Xinje XDPPro project, PLC1: RC2V6 (software 3.3 2016-03-11)

PROGRAM Ladder

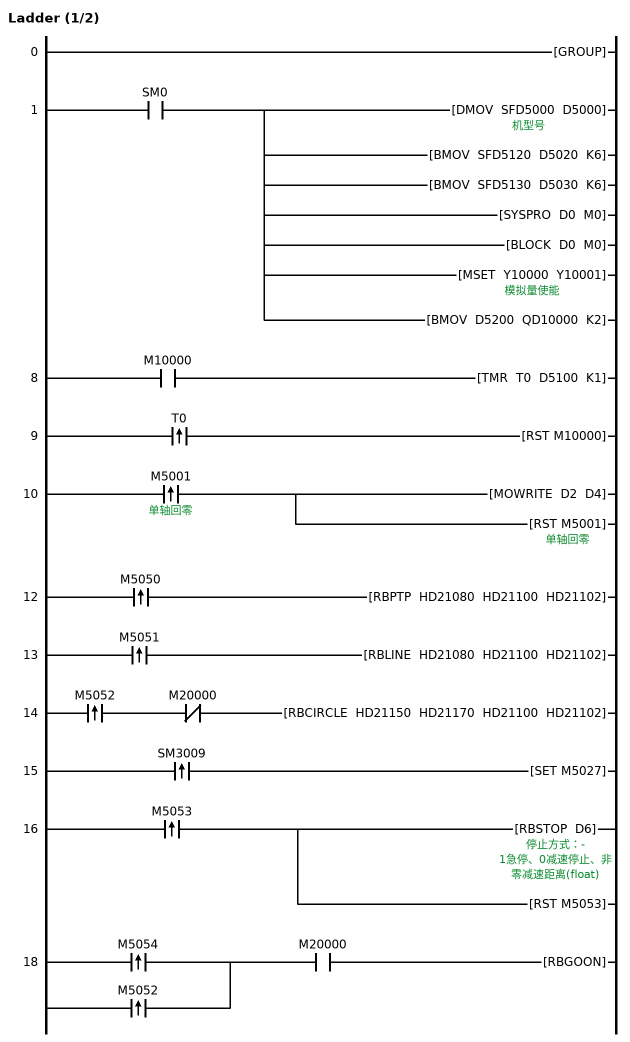
GROUP
LD     SM0
DMOV   SFD5000 D5000	; 机型号
BMOV   SFD5120 D5020 K6
BMOV   SFD5130 D5030 K6
SYSPRO D0 M0
BLOCK  D0 M0
MSET   Y10000 Y10001	; 模拟量使能
BMOV   D5200 QD10000 K2
LD     M10000
TMR    T0 D5100 K1
LDP    T0
RST    M10000
LDP    M5001	; 单轴回零
MOWRITE D2 D4
RST    M5001	; 单轴回零
LDP    M5050
RBPTP  HD21080 HD21100 HD21102
LDP    M5051
RBLINE HD21080 HD21100 HD21102
LDP    M5052
ANI    M20000
RBCIRCLE HD21150 HD21170 HD21100 HD21102
LDP    SM3009
SET    M5027
LDP    M5053
RBSTOP D6	; 停止方式：-1急停、0减速停止、非零减速距离(float)
RST    M5053
LDP    M5054
ORP    M5052
AND    M20000
RBGOON

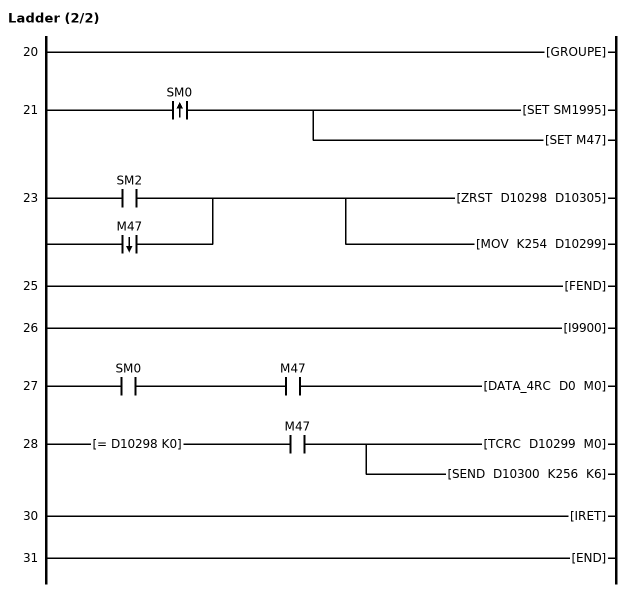
GROUPE
LDP    SM0
SET    SM1995
SET    M47
LD     SM2
ORF    M47
ZRST   D10298 D10305
MOV    K254 D10299
FEND
I9900
LD     SM0
AND    M47
DATA_4RC D0 M0
LD=    D10298 K0
AND    M47
TCRC   D10299 M0
SEND   D10300 K256 K6
IRET
END

COMMENTS (devices not used above)
M5040	PTP运动标志
HD0	shang
HD20	xia
HD40	chang
HD60	zhong
HD110	.

C FUNCTION BLOCK block.fcb
/*************************************************************************
   FunctionBlockName:  BLOCK
   Version:            1.0.0
   Author:             
   UpdateTime:         2016/6/1 9:27:03
   Comment:            
			20161123：RBON
**************************************************************************/
#define SysRegAddr_HD_SD_FD_SM_HSD_Y_X_D
#define PT_SIZE_WD          20
#define INT_BEGADDR_HD(i)   (10+i*2)       //200个int变量(10~309)
#define FLOAT_BEGADDR_HD(i) (410+i*2)      //200个float变量(410~809) 
#define POINT_BEGADDR_HD(i) (1000+i*PT_SIZE_WD)
#define Decimal_HEX(i)      (i-i/10*2)
#define SysModelType    X[26]          //0手动、1自动

//FUNC CODE
#define IF_BIT    1004
#define END_IF    1005
#define WAIT      1006
#define SET       1007
#define RESET     1008
#define IF_VALUE  1044
#define DELAY_MM  1003
#define LOOP      1009
#define END_LOOP  1010
#define WHILE     1011
#define END_WHILE 1012
#define LABLE     1013
#define GOTO      1014
#define ASSIGN    1020
#define PTASSIGN  1021
#define OFST      1022
#define SETACC    1023
#define CALL      1050
#define PTP       1030
#define MOVL      1031
#define MOVC      1032
#define WELD      1040
#define END_WELD  1041

#define MAINPRO_SIZE HD[3000]
#define SUBPRO1_SIZE HD[3001]
#define SUBPRO2_SIZE HD[3002]
#define SUBPRO3_SIZE HD[3003]
#define SUBPRO4_SIZE HD[3004]
#define TASK1_SIZE  HD[3005]
#define TASK2_SIZE  HD[3006]
#define proBlockSize(i) HD[3000+i]
#define SUBPRO_TOTAL_SIZE_WD 2000
#define FUNCCODE_SIZE_WD    20
#define MAINPRO_BEGADDR_HD  3020
#define SUBPRO_BEGADDR_HD   9020
#define curRunProIndex     HD[21040]
#define runRow_CurIndex(i) HD[21050+i]
#define runRow_UpIndex(i)  HD[21060+i]

#define X_BASE_BEGADDR  2140000000
#define Y_BASE_BEGADDR  2141000000
#define M_BASE_BEGADDR  2142000000
#define CHECK_X(index)  (index>=X_BASE_BEGADDR && index<=2140000099)
#define CHECK_Y(index)  (index>=Y_BASE_BEGADDR && index<=2141000199)
#define CHECK_M(index)  (index>=M_BASE_BEGADDR && index<=2142002999)

#define PRO_SINGLE_STEP_M 5025
#define PRO_RUN_M         5026
#define MOVE_END_FLAG     5027

#define PTP_TRIG_SINGAL_M    5050
#define MOVL_TRIG_SINGAL_M   5051
#define MOVC_TRIG_SINGAL_M   5052
#define ROBOT_RUNSTOP_M      5024

#define PT_BEGADDR_HD        21080
#define MOVSPEED_BEGADDR_HD  21100
#define MOVC_PT_BEGADDR_HD   21150
#define MOVC_PT_ENDADDR_HD   21170

#define ROBOT_ON   SM[3000]
#define RBRUN_ON   SM[3001]
#define ALARM_FLAG SM[3004]
#define WARN_FLAG  SM[3005]

#define ACCDEF_VALUE 70
#define SETACC_VALUE *(float*)&HD[21102]

float userSetAcc = 0;
int tmrVal=0;
int funcBegAddr_HD = 0;
int flag = 0,flag1=0;
extern int funcCodeRunFlag;
void funcExplanPro(BIT B,WORD W,int proIndex,int funcBegAddr_HD);
void IF_BIT_Pro(WORD W,BIT B,int pIndex);
void END_IF_Pro(int pIndex);
void DELAY_Pro(BIT B,WORD W,int proIndex);
void WAIT_Pro(BIT B,WORD W,int proIndex);
void SET_Pro(BIT B,int pIndex);
void RESET_Pro(BIT B,int pIndex);
void LOOP_Pro(int pIndex);
void END_LOOP_Pro(int pIndex);
void WHILE_Pro(WORD W,BIT B,int pIndex);
void END_WHILE_Pro(int pIndex);
void ASSIGN_Pro(WORD W,int pIndex);
void PTASSIGN_Pro(WORD W,int pIndex);
void OFST_Pro(WORD W,int pIndex);
void SETACC_Pro(WORD W,BIT B,int proIndex);
void GOTO_Pro(int pIndex);
void CALL_Pro();
void PTP_MOVL_Pro(BIT B,int proIndex);
void MOVC_Pro(BIT B,int proIndex);
void WELD_Pro(WORD W,BIT B,int proIndex);
void END_WELD_Pro(WORD W,BIT B,int proIndex);

#define RUNINDEX_PRO(proIndex){runRow_UpIndex(proIndex) = runRow_CurIndex(proIndex);\
					 runRow_CurIndex(proIndex)++;\
					 funcCodeRunFlag = 0;}

void BLOCK( WORD W , BIT B )
{
#define SysRegAddr_HD_SD_FD_SM_HSD_Y_X
#define DHD *(int*)&HD
#define FHD *(float*)&HD

	int i;
//B[10]=funcCodeRunFlag;
//B[11]=flag;
//B[12]=flag1;
	B[5056]=funcCodeRunFlag;
	if(userSetAcc==0)
		userSetAcc = ACCDEF_VALUE;	
	for(i=0; i<7; i++)
	{
		if(runRow_CurIndex(i)==0)
		{
			runRow_CurIndex(i)=1;
			flag = 0,flag1=0,funcCodeRunFlag = 0;
		}
	}
	if(ROBOT_ON==0||ALARM_FLAG==1||WARN_FLAG==1)
	{
		B[PTP_TRIG_SINGAL_M]=0;
		B[MOVL_TRIG_SINGAL_M]=0;
		B[MOVC_TRIG_SINGAL_M]=0;
		B[PRO_RUN_M]=0;
		flag = 0,flag1=0,funcCodeRunFlag = 0;
		B[MOVE_END_FLAG]=SM[3009];
		B[10000]=0;
		B[20000]=0;
		B[20001]=0;
		return;
	}
	if((B[PRO_SINGLE_STEP_M]==1||B[PRO_RUN_M]==1)&&B[20001]==1)
    	B[20001]=0;//清除圆弧未完成停止辅助信号
	if(runRow_CurIndex(curRunProIndex)<=proBlockSize(curRunProIndex)&&ALARM_FLAG==0)
	{
		if((B[PRO_SINGLE_STEP_M]==1||B[PRO_RUN_M]==1)&&funcCodeRunFlag==0)//下一步
		{
			funcCodeRunFlag=1;
			B[PRO_SINGLE_STEP_M]=0;
		}
	}
	if(funcCodeRunFlag==1)
	{
		funcBegAddr_HD = MAINPRO_BEGADDR_HD+(runRow_CurIndex(0)-1)*FUNCCODE_SIZE_WD;
		funcExplanPro(B,W,0,funcBegAddr_HD);
	}
}

void funcExplanPro(BIT B,WORD W,int proIndex,int funcBegAddr_HD)
{
	switch(HD[funcBegAddr_HD])
	{
	case IF_BIT:
		IF_BIT_Pro(W,B,proIndex);
		break;
	case END_IF:
		END_IF_Pro(proIndex);
		break;
	case DELAY_MM:
		DELAY_Pro(B,W,proIndex);
		break;
	case WAIT:
		WAIT_Pro(B,W,proIndex);
		break;
	case SET:
		SET_Pro(B,proIndex);
		break;
	case RESET:
		RESET_Pro(B,proIndex);
		break;
	case LOOP:
		LOOP_Pro(proIndex);
		break;
	case END_LOOP:
		END_LOOP_Pro(proIndex);
		break;
	case WHILE:
		WHILE_Pro(W,B,proIndex);
		break;
	case END_WHILE:
		END_WHILE_Pro(proIndex);
		break;
	case ASSIGN:
		ASSIGN_Pro(W,proIndex);
		break;
	case PTASSIGN:
		PTASSIGN_Pro(W,proIndex);
		break;
	case OFST:
		OFST_Pro(W,proIndex);
		break;
	case SETACC:
		SETACC_Pro(W,B,proIndex);
		break;	
	case LABLE:
		funcCodeRunFlag=0;
		runRow_UpIndex(proIndex) = runRow_CurIndex(proIndex);
		runRow_CurIndex(proIndex)++;
		break;
	case GOTO:
		GOTO_Pro(proIndex);
		break;
	case CALL:
		curRunProIndex = HD[funcBegAddr_HD+1];		
		CALL_Pro(B,W);
		break;
	case PTP:
		PTP_MOVL_Pro(B,proIndex);
		break;
	case MOVL:
		PTP_MOVL_Pro(B,proIndex);
		break;
	case MOVC:
		MOVC_Pro(B,proIndex);
		break;
	case WELD:
		WELD_Pro(W,B,proIndex);
		break;	
	case END_WELD:
		END_WELD_Pro(W,B,proIndex);
		break;	
	default:
		break;
	}
}

BOOL GetBitStatu(int bitAddr,BIT B)
{
	BOOL rlt=0;
	if(CHECK_X(bitAddr))
	{
		rlt = X[Decimal_HEX((bitAddr-X_BASE_BEGADDR))];
	}
	else if(CHECK_Y(bitAddr))
	{
		rlt = Y[Decimal_HEX((bitAddr-Y_BASE_BEGADDR))];
	}
	else if(CHECK_M(bitAddr))
	{
		rlt = B[bitAddr-M_BASE_BEGADDR];
	}
	return rlt;
}

BOOL GetBitCaseValue(BIT B,int begAddr)
{
	char cmpVal = 0;
	int para1 = DHD[begAddr+2],para2 = DHD[begAddr+4];
	int para3 = DHD[begAddr+6],para4 = DHD[begAddr+8];
	int para5 = DHD[begAddr+10],para6 = DHD[begAddr+12];
	int para7 = DHD[begAddr+14];
	
	cmpVal = GetBitStatu(para1,B);
	if(para2!=0)
	{
		if(para2==1)
			cmpVal = cmpVal|GetBitStatu(para3,B);
		else
			cmpVal = cmpVal&GetBitStatu(para3,B);
		if(para4!=0)
		{
			if(para4==1)
				cmpVal = cmpVal|GetBitStatu(para5,B);
			else
				cmpVal = cmpVal&GetBitStatu(para5,B);
			if(para6!=0)
			{
				if(para6==1)
					cmpVal = cmpVal|GetBitStatu(para7,B);
				else
					cmpVal = cmpVal&GetBitStatu(para7,B);
			}
		}
	}
	return cmpVal;
}

BOOL GetWordCompareResult(WORD W,int begAddr)
{
	char i,cmpVal = 0;
	float cmp[2]= {0};

	for(i=0; i<2; i++)
	{
		if(DHD[begAddr+4+i*6]==1)      //W
			cmp[i] = DHD[INT_BEGADDR_HD(DHD[begAddr+6+i*6])];
		else if(DHD[begAddr+4+i*6]==2) //F
			cmp[i] = FHD[FLOAT_BEGADDR_HD(DHD[begAddr+6+i*6])];
		else
			cmp[i] = FHD[begAddr+6+i*6];
	}
	if(DHD[begAddr+8]==1)
		cmpVal = (cmp[0]>cmp[1]);
	else if(DHD[begAddr+8]==2)
		cmpVal = (cmp[0]>=cmp[1]);
	else if(DHD[begAddr+8]==3)
		cmpVal = (cmp[0]<cmp[1]);
	else if(DHD[begAddr+8]==4)
		cmpVal = (cmp[0]<=cmp[1]);
	else if(DHD[begAddr+8]==5)
		cmpVal = (cmp[0]==cmp[1]);
	else if(DHD[begAddr+8]==6)
		cmpVal = (cmp[0]!=cmp[1]);
	return cmpVal;
}

void Set_Reset_Bit(BIT B,int addr,int value)
{
	int para1 = DHD[addr+2],para2 = DHD[addr+4];
	int i,index1,index2;
	if(CHECK_Y(para1))
	{
		index1 = para1-Y_BASE_BEGADDR;
		Y[Decimal_HEX(index1)]=value;
	}
	else if(CHECK_M(para1))
	{
		index1 = para1-M_BASE_BEGADDR;
		B[index1]=value;
	}
	if(para2!=0)
	{
		if(CHECK_Y(para2))
		{
			index2 = para2-Y_BASE_BEGADDR;
			for(i=0; i<(index2-index1+1); i++)
				Y[Decimal_HEX((index1+i))]=value;
		}
		else if(CHECK_M(para2))
		{
			index2=para2-M_BASE_BEGADDR;
			for(i=0; i<(index2-index1+1); i++)
				B[index1+i]=value;
		}
	}
}
float GetAssignPara(int type,int index,int addr)
{
	float val = 0;
	if(type==1)     //W
		val=DHD[INT_BEGADDR_HD(index)];
	else if(type==2)//F
		val=FHD[FLOAT_BEGADDR_HD(index)];
	else              //K
		val=FHD[funcBegAddr_HD+addr];
	return val;
}
float CalcAssignResult(int operateType,float para1,float para2)
{
	float val=0;
	if(operateType==1)
		val=para1+para2;
	else if(operateType==2)
		val=para1-para2;
	else if(operateType==3)
		val=para1*para2;
	else if(operateType==4)
		val=para1/para2;
	else
		val = para1;
	return val;
}

void DELAY_Pro(BIT B,WORD W,int proIndex)
{
	int type = HD[funcBegAddr_HD+1];
	if(flag==0)
	{
		if(type==0)
			DW[5100]=DHD[funcBegAddr_HD+2];
		else
			DW[5100]=DHD[INT_BEGADDR_HD(HD[funcBegAddr_HD+2])];
		if(DW[5100]!=0)
		{
			flag = 1;
			B[10000]=1;
		}
		else
		{
			flag = 0;
			funcCodeRunFlag=0;
			B[10000]=0;
		}
	}
	else if(flag==1&&B[10000]==0)
	{
		flag = 0;
		RUNINDEX_PRO(proIndex)
	}
}

void IF_BIT_Pro(WORD W,BIT B,int proIndex)
{
	BOOL tmpBL = 0;
	if(DHD[funcBegAddr_HD+2]>=X_BASE_BEGADDR)
		tmpBL = GetBitCaseValue(B,funcBegAddr_HD);
	else
		tmpBL=GetWordCompareResult(W,funcBegAddr_HD);

	if(tmpBL==1)
	{
		RUNINDEX_PRO(proIndex)
	}
	else
	{
		int j,cycNum = proBlockSize(proIndex)-runRow_CurIndex(proIndex);
		for(j=0; j<cycNum; j++)
		{
			int tmpFuncCode = HD[funcBegAddr_HD+(j+1)*FUNCCODE_SIZE_WD];
			int endFlag = HD[funcBegAddr_HD+(j+1)*FUNCCODE_SIZE_WD+1];
			if(tmpFuncCode==END_IF&&endFlag==runRow_CurIndex(proIndex))
			{
				runRow_CurIndex(proIndex) = runRow_CurIndex(proIndex)+j+1;
				funcCodeRunFlag = 0;
				break;
			}
		}
	}
}
void END_IF_Pro(int proIndex)
{
	RUNINDEX_PRO(proIndex)
}

void WAIT_Pro(BIT B,WORD W,int proIndex)
{
	int timeType = DHD[funcBegAddr_HD+15],timeVal = DHD[funcBegAddr_HD+17];
	int fltTime = HD[funcBegAddr_HD+19],blTmp=0;
	int blrslt=0;
	int siglRslt = GetBitCaseValue(B,funcBegAddr_HD-1);
	
	if(timeType!=0)
		timeVal = DHD[INT_BEGADDR_HD(timeVal)];
	if(fltTime!=0&&siglRslt==1&&flag1==0)
	{		
		if(flag==1&&SM[11]==0)
			tmrVal++;
		flag = SM[11];
		if(tmrVal*5<fltTime)
			return;	
	}
	else
		flag1 = 1;
			
	if(timeVal!=0 && flag1==1 && flag==0)
	{
		DW[5100]=timeVal;
		B[10000]=1;	
		flag = 1;
	}
	if(timeVal!=0&&flag1==1&&B[10000]==0)
	{
		blTmp = 1;	
		flag = 0;
	}
	if(siglRslt==1 || blTmp==1)
	{
		RUNINDEX_PRO(proIndex)		
	}
	tmrVal = 0;
	flag1 = 0;
}
void SET_Pro(BIT B,int proIndex)
{
	Set_Reset_Bit(B,funcBegAddr_HD,1);
	RUNINDEX_PRO(proIndex)
}
void RESET_Pro(BIT B,int proIndex)
{
	Set_Reset_Bit(B,funcBegAddr_HD,0);
	RUNINDEX_PRO(proIndex)
}

void LOOP_Pro(int proIndex)
{
	int para1=DHD[funcBegAddr_HD+2],para2=DHD[funcBegAddr_HD+4];
	int loop_cycNum=0,begAddr=0;
	if(para1==0)
		loop_cycNum = para2;
	else
		loop_cycNum = DHD[INT_BEGADDR_HD(para2)];
	if(proIndex==0)
		begAddr=MAINPRO_BEGADDR_HD;
	else
		begAddr=SUBPRO_BEGADDR_HD;
	if(runRow_CurIndex(proIndex)>=runRow_UpIndex(proIndex))//||HD[begAddr+(runRow_UpIndex(proIndex)-1)*FUNCCODE_SIZE_WD]!=END_LOOP)
		DHD[funcBegAddr_HD+8]=0;

	if(loop_cycNum<=0)
	{
		int j,cycNum = proBlockSize(proIndex)-runRow_CurIndex(proIndex);
		for(j=0; j<cycNum; j++)
		{
			int tmpFuncCode = HD[funcBegAddr_HD+(j+1)*FUNCCODE_SIZE_WD];
			int endFlag = HD[funcBegAddr_HD+(j+1)*FUNCCODE_SIZE_WD+1];
			if(tmpFuncCode==END_LOOP&&endFlag==runRow_CurIndex(proIndex))
			{
				runRow_CurIndex(proIndex) = runRow_CurIndex(proIndex)+j+1;
				break;
			}
		}
	}
	else
	{
		DHD[funcBegAddr_HD+8]=DHD[funcBegAddr_HD+8]+1;
		RUNINDEX_PRO(proIndex)
	}
	funcCodeRunFlag = 0;
}
void END_LOOP_Pro(int proIndex)
{
	int para1=DHD[funcBegAddr_HD+1];
	int loop_BegAddr=0,loop_para1,loop_para2,curNum,loop_cycNum=0;
	if(proIndex==0)
		loop_BegAddr = MAINPRO_BEGADDR_HD+(para1-1)*FUNCCODE_SIZE_WD;
	else
		loop_BegAddr = SUBPRO_BEGADDR_HD+(proIndex-1)*SUBPRO_TOTAL_SIZE_WD+(para1-1)*FUNCCODE_SIZE_WD;

	loop_para1=DHD[loop_BegAddr+2];
	loop_para2=DHD[loop_BegAddr+4];
	curNum = DHD[loop_BegAddr+8];

	if(loop_para1==0)
		loop_cycNum = loop_para2;
	else
		loop_cycNum = DHD[INT_BEGADDR_HD(loop_para2)];

	runRow_UpIndex(proIndex) = runRow_CurIndex(proIndex);
	if(curNum==loop_cycNum)
	{
		DHD[loop_BegAddr+8]=0;
		runRow_CurIndex(proIndex)++;
	}
	else
		runRow_CurIndex(proIndex)=para1;
	funcCodeRunFlag = 0;
}
void WHILE_Pro(WORD W,BIT B,int proIndex)
{
	BOOL tmpBL = 0;
	if(DHD[funcBegAddr_HD+2]>=X_BASE_BEGADDR)
		tmpBL = GetBitCaseValue(B,funcBegAddr_HD);
	else
		tmpBL=GetWordCompareResult(W,funcBegAddr_HD);
	if(tmpBL==1)
	{
		RUNINDEX_PRO(proIndex)
	}
	else
	{
		int j,cycNum = proBlockSize(proIndex)-runRow_CurIndex(proIndex);
		for(j=0; j<cycNum; j++)
		{
			int tmpFuncCode = HD[funcBegAddr_HD+(j+1)*FUNCCODE_SIZE_WD];
			int endFlag = HD[funcBegAddr_HD+(j+1)*FUNCCODE_SIZE_WD+1];
			if(tmpFuncCode==END_WHILE&&endFlag==runRow_CurIndex(proIndex))
			{
				runRow_CurIndex(proIndex) = runRow_CurIndex(proIndex)+j+1+1;
				funcCodeRunFlag = 0;
				break;
			}
		}
	}
}
void END_WHILE_Pro(int proIndex)
{
	int para1=DHD[funcBegAddr_HD+1];

	runRow_UpIndex(proIndex) = runRow_CurIndex(proIndex);
	runRow_CurIndex(proIndex) = para1;
	funcCodeRunFlag = 0;
}

void ASSIGN_Pro(WORD W,int proIndex)
{
	int leftParaType = HD[funcBegAddr_HD+1],leftPara=HD[funcBegAddr_HD+2];

	int rightPara1Type = DHD[funcBegAddr_HD+4],rightPara1=DHD[funcBegAddr_HD+6];
	int operaFlag1 = DHD[funcBegAddr_HD+8];
	int rightPara2Type = DHD[funcBegAddr_HD+10],rightPara2=DHD[funcBegAddr_HD+12];
	int operaFlag2 = DHD[funcBegAddr_HD+14];
	int rightPara3Type = DHD[funcBegAddr_HD+16],rightPara3=DHD[funcBegAddr_HD+18];

	float result1,result;
	float para1=GetAssignPara(rightPara1Type,rightPara1,6);
	float para2=GetAssignPara(rightPara2Type,rightPara2,12);
	float para3=GetAssignPara(rightPara3Type,rightPara3,18);

	result1 = CalcAssignResult(operaFlag1,para1,para2);
	result = CalcAssignResult(operaFlag2,result1,para3);

	if(leftParaType==1)
		DHD[INT_BEGADDR_HD(leftPara)]=result;
	else if(leftParaType==2)
		FHD[FLOAT_BEGADDR_HD(leftPara)]=result;
	RUNINDEX_PRO(proIndex)
}

void PTASSIGN_Pro(WORD W,int proIndex)
{
	int targetPtType = HD[funcBegAddr_HD+1],targetPt=0;
	int basePtType =   HD[funcBegAddr_HD+3],basePt=0;
	int coordIndex =   HD[funcBegAddr_HD+5];
	int ofstValueType1 =HD[funcBegAddr_HD+7],ofstValue1=DHD[funcBegAddr_HD+8];
	int operaFlag1 = HD[funcBegAddr_HD+10];	
	int ofstValueType2 =HD[funcBegAddr_HD+11],ofstValue2=DHD[funcBegAddr_HD+12];
	float para1=0,para2=0,ofstValue=0;
	para1=GetAssignPara(ofstValueType1,ofstValue1,8);
	if(operaFlag1!=0)
		para2=GetAssignPara(ofstValueType2,ofstValue2,12);
	ofstValue = CalcAssignResult(operaFlag1,para1,para2);
	if(targetPtType==0)
		targetPt = HD[funcBegAddr_HD+2];
	else
		targetPt = DHD[INT_BEGADDR_HD(HD[funcBegAddr_HD+2])];
	if(basePtType==0)
		basePt = HD[funcBegAddr_HD+4];
	else
		basePt = DHD[INT_BEGADDR_HD(HD[funcBegAddr_HD+4])];			  		
	memcpy(HD+POINT_BEGADDR_HD(targetPt),HD+POINT_BEGADDR_HD(basePt),20*2);

	if(coordIndex==4)
		coordIndex = 6; //RZ
	FHD[POINT_BEGADDR_HD(targetPt)+(coordIndex-1)*2] = FHD[POINT_BEGADDR_HD(basePt)+(coordIndex-1)*2] + ofstValue;
	RUNINDEX_PRO(proIndex)
}

void OFST_Pro(WORD W,int proIndex)
{
	int i,targetPt = HD[funcBegAddr_HD+1],basePt=HD[funcBegAddr_HD+2];
	float ofstValueBuf=0;

	memcpy(HD+POINT_BEGADDR_HD(targetPt),HD+POINT_BEGADDR_HD(basePt),20*2);
	for(i=0; i<3; i++)
	{
		if(HD[funcBegAddr_HD+3+i*3]==0)
			ofstValueBuf = FHD[funcBegAddr_HD+4+i*3];
		else
			ofstValueBuf = DHD[INT_BEGADDR_HD(DHD[funcBegAddr_HD+4+i*3])];
		FHD[POINT_BEGADDR_HD(targetPt)+i*2] = FHD[POINT_BEGADDR_HD(basePt)+i*2]+ofstValueBuf;
	}
	RUNINDEX_PRO(proIndex)
}

float SETACC_between;
void SETACC_Pro(WORD W,BIT B,int proIndex)
{
	int type = HD[funcBegAddr_HD+1];
	int value = DHD[funcBegAddr_HD+2];
	int flag = DHD[funcBegAddr_HD+4];
	if(type!=0)
		value=DHD[INT_BEGADDR_HD(HD[funcBegAddr_HD+2])];
	if(flag==1)	
		userSetAcc = value;
	else
	{
		SETACC_VALUE = value;	
	    SETACC_between=value;
	}
	RUNINDEX_PRO(proIndex)
}

void WELD_Pro(WORD W,BIT B,int proIndex)
{
	int type_V = HD[funcBegAddr_HD+1],type_A = HD[funcBegAddr_HD+4];
	float value_V = FHD[funcBegAddr_HD+2],value_A = FHD[funcBegAddr_HD+5];

	if(type_V!=0)
		value_V=DHD[INT_BEGADDR_HD(HD[funcBegAddr_HD+2])];
	if(type_A!=0)
		value_A=DHD[INT_BEGADDR_HD(HD[funcBegAddr_HD+5])];	
			
	W[5201] = (value_V-2)/0.02;
	W[5200] = (value_A-80)/0.1;	
	
	//if(B[10000]==0)
	{
		//B[10000]=1;
		//W[5100]=200;//延时200MS
	}
	if(B[10000]==0)
	{
		B[10000]=1;
		W[5100]=200;//延时200MS
		if(B[5101]==0)//模拟焊关闭
			Y[8]=1;
		RUNINDEX_PRO(proIndex)
	}
}

void END_WELD_Pro(WORD W,BIT B,int proIndex)
{
	Y[8]=0;
	RUNINDEX_PRO(proIndex)
}

void GOTO_Pro(int proIndex)
{
	int i,jumpTargetIndex = HD[funcBegAddr_HD+1];
	int cycNum = 0,begAddr=0;
	
	if(proIndex==0)
		cycNum = MAINPRO_SIZE;
	else if(proIndex==1)
		cycNum = SUBPRO1_SIZE;
	else if(proIndex==2)
		cycNum = SUBPRO2_SIZE;
	else if(proIndex==3)
		cycNum = SUBPRO3_SIZE;
	else if(proIndex==4)
		cycNum = SUBPRO4_SIZE;
	if(proIndex==0)
		begAddr = MAINPRO_BEGADDR_HD;
	else
		begAddr = SUBPRO_BEGADDR_HD+(proIndex-1)*SUBPRO_TOTAL_SIZE_WD;				
		
	runRow_UpIndex(proIndex) = runRow_CurIndex(proIndex);
	for(i=0;i<cycNum;i++)
	{
		int funcCode = HD[begAddr+i*20],jumpIndex=HD[begAddr+i*20+1];
		if(funcCode==LABLE&&jumpIndex==jumpTargetIndex)
		{
			runRow_CurIndex(proIndex)=i+1;
			break;
		}
	}
	funcCodeRunFlag = 0;
}

void CALL_Pro(BIT B,WORD W)
{
	int	pIndex = HD[funcBegAddr_HD+1];

	if(flag1==1)
	{
		funcBegAddr_HD = SUBPRO_BEGADDR_HD+(runRow_CurIndex(pIndex)-1)*FUNCCODE_SIZE_WD+(pIndex-1)*SUBPRO_TOTAL_SIZE_WD;
		funcExplanPro(B,W,pIndex,funcBegAddr_HD);
	}
	else
	{
		flag1 = 1;
		funcCodeRunFlag=0;
	}
	if(runRow_CurIndex(pIndex)==(proBlockSize(pIndex)+1))
	{
		runRow_CurIndex(pIndex)=1;
		runRow_CurIndex(0)++;
		curRunProIndex = 0;
		flag1 = 0;
	}
}

void PTP_MOVL_Pro(BIT B,int proIndex)
{
	float psdPer = 0,zone=0;;
	int ptNum;
	int funcCode = HD[funcBegAddr_HD+0];
	
	if(HD[funcBegAddr_HD+1]==0)
		ptNum = DHD[funcBegAddr_HD+2];
	else
		ptNum = DHD[INT_BEGADDR_HD(DHD[funcBegAddr_HD+2])];	
	if((funcCode==PTP ? B[PTP_TRIG_SINGAL_M]==1 : B[MOVL_TRIG_SINGAL_M]==1)&&B[MOVE_END_FLAG]==1)
	{
		RUNINDEX_PRO(proIndex)
		B[PTP_TRIG_SINGAL_M]=0;
		B[MOVL_TRIG_SINGAL_M]=0;
	}
	else if(B[MOVE_END_FLAG]==1)
	{
		if(HD[funcBegAddr_HD+4]==0)
			psdPer = *(float*)&HD[funcBegAddr_HD+5];
		else
			psdPer = DHD[INT_BEGADDR_HD(DHD[funcBegAddr_HD+5])];
		if(HD[funcBegAddr_HD+7]==0)
			zone = *(float*)&HD[funcBegAddr_HD+8];
		else
			zone = DHD[INT_BEGADDR_HD(DHD[funcBegAddr_HD+8])];
		memcpy(HD+PT_BEGADDR_HD,HD+POINT_BEGADDR_HD(ptNum),10*2*2);
		HD[PT_BEGADDR_HD+17]=zone;
		if(SysModelType==0)//手动
		{
		FHD[MOVSPEED_BEGADDR_HD]=psdPer;	
			if(HD[funcBegAddr_HD-FUNCCODE_SIZE_WD]!=SETACC||(HD[funcBegAddr_HD-FUNCCODE_SIZE_WD]==SETACC&&HD[funcBegAddr_HD-FUNCCODE_SIZE_WD+4]==1))
				SETACC_VALUE = userSetAcc*0.6;
			else
				SETACC_VALUE=SETACC_between*0.6;		
		}
		else//自动
		{
			FHD[MOVSPEED_BEGADDR_HD]=psdPer;	
			if(HD[funcBegAddr_HD-FUNCCODE_SIZE_WD]!=SETACC||(HD[funcBegAddr_HD-FUNCCODE_SIZE_WD]==SETACC&&HD[funcBegAddr_HD-FUNCCODE_SIZE_WD+4]==1))
				SETACC_VALUE = userSetAcc;		
		}
		if(funcCode==PTP)
			B[PTP_TRIG_SINGAL_M]=1;
		else
			B[MOVL_TRIG_SINGAL_M]=1;
		B[MOVE_END_FLAG]=0;
	}
}

void MOVC_Pro(BIT B,int proIndex)
{
	float psdPer = 0,zone=0;;
	int ptNum1,ptNum2;
	
	if(HD[funcBegAddr_HD+1]==0)
		ptNum1 = DHD[funcBegAddr_HD+2];
	else
		ptNum1 = DHD[INT_BEGADDR_HD(DHD[funcBegAddr_HD+2])];
		
	if(HD[funcBegAddr_HD+4]==0)
		ptNum2 = DHD[funcBegAddr_HD+5];
	else
		ptNum2 = DHD[INT_BEGADDR_HD(DHD[funcBegAddr_HD+5])];	
			
	if(B[MOVC_TRIG_SINGAL_M]==1&&B[MOVE_END_FLAG]==1)
	{
		RUNINDEX_PRO(proIndex)
		B[MOVC_TRIG_SINGAL_M]=0;
		B[20000]=0;//圆弧未完成停止标志
	}
	else if(B[MOVE_END_FLAG]==1 && B[20000]==0)
	{
		if(HD[funcBegAddr_HD+7]==0)
			psdPer = *(float*)&HD[funcBegAddr_HD+8];
		else
			psdPer = DHD[INT_BEGADDR_HD(DHD[funcBegAddr_HD+8])];
		if(HD[funcBegAddr_HD+10]==0)
			zone = *(float*)&HD[funcBegAddr_HD+11];
		else
			zone = DHD[INT_BEGADDR_HD(DHD[funcBegAddr_HD+11])];
		memcpy(HD+MOVC_PT_BEGADDR_HD,HD+POINT_BEGADDR_HD(ptNum1),10*2*2);
		memcpy(HD+MOVC_PT_ENDADDR_HD,HD+POINT_BEGADDR_HD(ptNum2),10*2*2);
		HD[MOVC_PT_ENDADDR_HD+17]=zone;
		FHD[MOVSPEED_BEGADDR_HD]=psdPer;
		B[MOVC_TRIG_SINGAL_M]=1;
		if(SysModelType==0)
		{
			if(HD[funcBegAddr_HD-FUNCCODE_SIZE_WD]!=SETACC||(HD[funcBegAddr_HD-FUNCCODE_SIZE_WD]==SETACC&&HD[funcBegAddr_HD-FUNCCODE_SIZE_WD+4]==1))
				SETACC_VALUE = userSetAcc*0.6;
			else
				SETACC_VALUE=SETACC_between*0.6;	
		}
		else
		{
			if(HD[funcBegAddr_HD-FUNCCODE_SIZE_WD]!=SETACC||(HD[funcBegAddr_HD-FUNCCODE_SIZE_WD]==SETACC&&HD[funcBegAddr_HD-FUNCCODE_SIZE_WD+4]==1))
				SETACC_VALUE = userSetAcc;
		}
		B[MOVE_END_FLAG]=0;
	}
	else if(B[20000]==1)
	{
		B[MOVC_TRIG_SINGAL_M]=1;
		B[MOVE_END_FLAG]=0;
	}
}

C FUNCTION BLOCK data_4rc.fcb
/* RC自由格式通讯 */
/*************************************************************************
   FunctionBlockName:  DATA_4RC
   Version:            1.0.0
   Author:             clm
   UpdateTime:         2016-1-22 15:31:37
   Comment:            
			自由格式通讯
**************************************************************************/
void DATA_4RC( WORD W , BIT B )
{
	#define SysRegAddr_HD_D_SD_HSD_SM
	
	int i=0,j=0;
	
	D[10300] = 0x0055;			//起始符1
	D[10301] = 0x0055;			//起始符2
	if(D[10298] == 0)					//单双周期判断
	{
		D[10302] = D[10302]+1;			//上周期数据序号
		if(D[10302]>=256)
		{
			D[10302] = 0;
			D[10303] = D[10303]+1;
		}
		if(D[10303]>=256)
		{
			D[10303] = 0;
			D[10304] = D[10304]+1;
		}
		if(D[10304]>=256)
		{
			D[10304] = 0;
			D[10305] = D[10305]+1;
		}
		if(D[10305]>=256)
		{
			D[10305] = 0;
		}		
		for(i=0;i<6;i++)
		{
			D[10306+16*i] = (*(INT16S*)&HSD[100+20*i]&0x00ff);		//轴n位置给定(n=1~6)
			D[10307+16*i] = (*(INT16S*)&HSD[100+20*i]&0xff00)>>8;
			D[10308+16*i] = (*(INT16S*)&HSD[101+20*i]&0x00ff);
			D[10309+16*i] = (*(INT16S*)&HSD[101+20*i]&0xff00)>>8;
			D[10310+16*i] = (*(INT16S*)&HSD[102+20*i]&0x00ff);
			D[10311+16*i] = (*(INT16S*)&HSD[102+20*i]&0xff00)>>8;
			D[10312+16*i] = (*(INT16S*)&HSD[103+20*i]&0x00ff);
			D[10313+16*i] = (*(INT16S*)&HSD[103+20*i]&0xff00)>>8;
			D[10314+16*i] = (*(INT16S*)&HSD[104+20*i]&0x00ff);		//轴n位置反馈
			D[10315+16*i] = (*(INT16S*)&HSD[104+20*i]&0xff00)>>8;
			D[10316+16*i] = (*(INT16S*)&HSD[105+20*i]&0x00ff);
			D[10317+16*i] = (*(INT16S*)&HSD[105+20*i]&0xff00)>>8;
			D[10318+16*i] = (*(INT16S*)&HSD[106+20*i]&0x00ff);
			D[10319+16*i] = (*(INT16S*)&HSD[106+20*i]&0xff00)>>8;
			D[10320+16*i] = (*(INT16S*)&HSD[107+20*i]&0x00ff);
			D[10321+16*i] = (*(INT16S*)&HSD[107+20*i]&0xff00)>>8;
		}
		for(i=0;i<24;i=i+2)
		{
			j=i/2;
			D[10402+i] = (*(INT16S*)&SD[4000+j]&0x00ff);			//空间坐标位置SD4000~4011
			D[10403+i] = (*(INT16S*)&SD[4000+j]&0xff00)>>8;
		}
		D[10426] = (*(INT16S*)&SD[4016]&0x00ff);					//坐标属性SD4016~4019
		D[10427] = (*(INT16S*)&SD[4016]&0xff00)>>8;
		D[10428] = (*(INT16S*)&SD[4017]&0x00ff);
		D[10429] = (*(INT16S*)&SD[4017]&0xff00)>>8;
		D[10430] = (*(INT16S*)&SD[4018]&0x00ff);
		D[10431] = (*(INT16S*)&SD[4018]&0xff00)>>8;
		D[10432] = (*(INT16S*)&SD[4019]&0x00ff);
		D[10433] = (*(INT16S*)&SD[4019]&0xff00)>>8;
		for(i=0;i<24;i=i+2)
		{
			j=i/2;
			D[10434+i] = (*(INT16S*)&SD[4020+j]&0x00ff);			//空间坐标位置SD4020~4031
			D[10435+i] = (*(INT16S*)&SD[4020+j]&0xff00)>>8;
		}
		for(i=0;i<24;i=i+2)
		{
			j=i/2;
			D[10458+i] = (*(INT16S*)&SD[4060+j]&0x00ff);			//空间坐标位置SD4060~4071
			D[10459+i] = (*(INT16S*)&SD[4060+j]&0xff00)>>8;
		}
		for(i=0;i<24;i=i+2)
		{
			j=i/2;
			D[10482+i] = (*(INT16S*)&SD[4080+j]&0x00ff);			//空间坐标位置SD4080~4091
			D[10483+i] = (*(INT16S*)&SD[4080+j]&0xff00)>>8;
		}
		for(i=0;i<24;i=i+2)
		{
			j=i/2;
			D[10506+i] = (*(INT16S*)&SD[4800+j]&0x00ff);			//空间坐标位置SD4800~4811(带工具反馈)
			D[10507+i] = (*(INT16S*)&SD[4800+j]&0xff00)>>8;
		}
		for(i=0;i<24;i=i+2)
		{
			j=i/2;
			D[10530+i] = (*(INT16S*)&SD[4820+j]&0x00ff);			//空间坐标位置SD4820~4831(带工具给定)
			D[10531+i] = (*(INT16S*)&SD[4820+j]&0xff00)>>8;
		}
	}
	else
	{
		D[10298] = 0;
	}
	
}

C FUNCTION BLOCK syspro.fcb
/*************************************************************************
   FunctionBlockName:  SYSPRO
   Version:            1.0.0
   Author:             
   UpdateTime:         2016/6/12 12:46:52
   Comment:            
			20161126:
**************************************************************************/
#define DEVICETYPE *(int*)(W+5000)
#define AXISCNT 6
#define STOP_SIGNAL    (X[24]||X[25]) //试教器急停X30、控制柜急停X31
#define ENABLE_SIGNAL   X[1]
#define SysModelType    X[26]          //0手动、1自动
#define WELD_STOP {Y[8]=0;Y[9]=0;}     //焊接点火、送丝
#define SYS_LIGHT_Y  24                //系统指示灯Y30

#define ERR_CLEAR_FLAG_M 5020
#define ROBOT_ALARM_M    5021
#define ROBOT_STATUS_M   5022
#define ROBOT_ENABLE     B[5023]
#define ROBOT_RUNSTOP_M  5024

#define PTP_TRIG_SINGAL_M    5050
#define MOVL_TRIG_SINGAL_M   5051
#define MOVC_TRIG_SINGAL_M   5052
#define PRO_SINGLE_STEP_M    5025
#define PRO_RUN_M            5026

#define ERR_CODE_W       5010
#define SYSADMIN_CODE    W[5014]
#define Sys_StopModel(i) (FW[6]=i)

#define TOOLINDEX ((char)HD[21070])
#define REF_COORD_INDEX ((char)W[5011])
#define JOINT_COORD_INDEX 5
#define runRow_CurIndex(i) HD[21050+i]
#define runRow_UpIndex(i)  HD[21060+i]
#define ROBOT_ENABLE_SM     3040
#define JOINT_SIMULAT_SM(i) (2018+i*20)
#define JOINT_ENABLE_SM(i)  (2010+i*20)
#define ROBOT_ON_SM   3000
#define RBRUN_ON_SM   3001
#define ALARM_FLAG_SM 3004
#define WARN_FLAG_SM  3005

void sysRBON(WORD W,BIT B);
void jogProcess(WORD W,BIT B);
void sysStatusCheck(WORD W,BIT B);
void postionDisPlay(WORD W,BIT B);
void checkArea(WORD W,BIT B);
void round_area(WORD W,BIT B);//球形区域检测
void cylinder_area(WORD W,BIT B);//圆柱体

int jogFlagVal[6*2]= {0},edgeFlagVal[6*2]= {0};
int funcCodeRunFlag=0;
void SYSPRO( WORD W , BIT B )
{
#define SysRegAddr_HD_SD_FD_SM_HSD_Y_X_HM
               
	*((char*)(SD+4018)+0)=REF_COORD_INDEX; //低字节：参考坐标系
	*((char*)(SD+4018)+1)=TOOLINDEX;       //高字节：工具号(掉电保持)
	
	if(B[ROBOT_RUNSTOP_M]==1)
	{
		if(B[MOVC_TRIG_SINGAL_M]==1)
			B[20000]=1;//圆弧停止标志
		B[ROBOT_RUNSTOP_M]=0;
		Sys_StopModel(0);
		B[5026]=0;
		B[5053]=1;
		funcCodeRunFlag=0;
		B[PTP_TRIG_SINGAL_M]=0;
		B[MOVL_TRIG_SINGAL_M]=0;
		B[MOVC_TRIG_SINGAL_M]=0;
	}
#define between_flag   20001
	if(B[20000]==1||B[between_flag]==1)//在运行时判断是否改变指针位置
	{
		if((runRow_CurIndex(0)-runRow_UpIndex(0))!=1)//判断圆弧停止是否改变指针位置
			B[20000]=0;//改变指针后圆弧不在执RBGOON
		if((runRow_CurIndex(0)-runRow_UpIndex(0))==1)
			B[20000]=1;
		if(B[RBRUN_ON_SM]==0&&B[MOVC_TRIG_SINGAL_M]==0)
			B[between_flag]=1;
	}
	if(DEVICETYPE!=0)
	{
		sysStatusCheck(W,B);
		sysRBON(W,B);
		jogProcess(W,B);
		checkArea(W,B);
		round_area(W,B);//球
		cylinder_area(W,B);//圆柱体
	}
}

void sysRBON(WORD W,BIT B)
{
#define SysRegAddr_HD_SD_FD_SM_HSD_Y_X_HM
	int i;
	for(i=0; i<AXISCNT; i++)
		SM[JOINT_SIMULAT_SM(i)] = 1;
	if(STOP_SIGNAL==1&&((ENABLE_SIGNAL==1&&SysModelType==0)||(ROBOT_ENABLE==1&&SysModelType==1))&&B[ROBOT_ALARM_M]==0&&SYSADMIN_CODE==2)
	{
		//使能开启
		for(i=0; i<AXISCNT; i++)
			SM[JOINT_ENABLE_SM(i)]=1;
		if(SM[2000]==1&&SM[2020]==1&&SM[2040]==1&&SM[2060]==1&&SM[2080]==1&&SM[2100]==1&&SM[13]==1)
			SM[ROBOT_ENABLE_SM]=1;
	}
	else if(STOP_SIGNAL==0||(ENABLE_SIGNAL==0&&SysModelType==0)||(ROBOT_ENABLE==0&&SysModelType==1)||B[ROBOT_ALARM_M]==1||(ROBOT_ENABLE==1&&SysModelType==0))
	{
		//使能关闭
		B[5023] = 0;
		WELD_STOP;//关闭送丝及焊枪点火
		for(i=0; i<AXISCNT; i++)
			SM[JOINT_ENABLE_SM(i)]=0;
		if(SM[2000]==0&&SM[2020]==0&&SM[2040]==0&&SM[2060]==0&&SM[2080]==0&&SM[2100]==0)
			SM[ROBOT_ENABLE_SM]=0;
		for(i=0; i<AXISCNT; i++)
		{
			edgeFlagVal[0+i*2]=0;
			edgeFlagVal[1+i*2]=0;
			jogFlagVal[0+i*2]=0;
			jogFlagVal[1+i*2]=0;
		}
	}
	if(SM[ROBOT_ON_SM]==1&&SM[ALARM_FLAG_SM]==0&&SM[WARN_FLAG_SM]==0&&B[ROBOT_ALARM_M]==0)
		B[ROBOT_STATUS_M]=1;
	else
		B[ROBOT_STATUS_M]=0;
}

void sysStatusCheck(WORD W,BIT B)
{
#define SysRegAddr_HD_SD_FD_SM_HSD_Y_X_HM
#define DSD *(int*)&SD

	int i,j,k[AXISCNT]= {0};
	int commErrCnt[AXISCNT]= {0};
	if(B[ERR_CLEAR_FLAG_M]==1)//清除报警
	{
		W[ERR_CODE_W] =0;
		B[ROBOT_ALARM_M]=0;
		SM[ALARM_FLAG_SM]=0;
		SM[WARN_FLAG_SM]=0;
		for(i=0; i<AXISCNT; i++)
		{
			SM[2004+i*60]=0;
			DSD[2002+i*60]=0;
		}
		DSD[4130]=0;
		B[ERR_CLEAR_FLAG_M]=0;
		return;
	}

	for(i=0; i<AXISCNT; i++)
	{
		for(j=0; j<5; j++)
		{
			if((DSD[2004+i*60]-commErrCnt[i])>=1)
				k[i]++;
		}
		commErrCnt[i]=DSD[2004+i*60];
		if(k[i]==5&&SM[2004+i*20]==1&&SD[2002+i*60]==20011)
		{
			W[ERR_CODE_W]=20+i;
			break;
		}
	}
	if(STOP_SIGNAL==0)//急停
	{
		W[ERR_CODE_W]=26;
	}
	else if(SM[ALARM_FLAG_SM]==1)
	{
		W[ERR_CODE_W]=SD[4130];
	}
	else if(SM[WARN_FLAG_SM]==1)
	{
		W[ERR_CODE_W]=SD[4131];
	}

	if(W[ERR_CODE_W]==0)//报警指示灯
		Y[SYS_LIGHT_Y]=1;//正常：常亮
	else
	{
		B[ROBOT_ALARM_M]=1;
		if(SM[13]==0)//报警：闪烁(1s)
			Y[SYS_LIGHT_Y]=0;
		else
			Y[SYS_LIGHT_Y]=1;
	}
}

void jogProcess(WORD W,BIT B)
{
#define SysRegAddr_HD_SD_FD_SM_HSD_Y_X_HM
#define FHD *(float*)&HD
#define FSD *(float*)&SD
#define DSD *(int*)&SD

#define AxisJogStep FSD[4110]
#define AxisJogSpeed DSD[4112]
#define AxisJogSpeed_SET DW[5032]

#define CoordJogStep FSD[4100]
#define CoordJogSpeed DSD[4102]
#define CoordJogSpeed_SET DW[5022]

#define UserDefSpeed FHD[21072]
#define GAPVALUE 10

#define COORD_JOG_SM(i) (3050+i)
#define JOINT_JOG_SM(i) (3070+i)

	int i,j,index=0,flag = 0;
	if(SM[ROBOT_ON_SM]==0||SM[ALARM_FLAG_SM]==1)
		return;
	if(UserDefSpeed==0)
		UserDefSpeed = 10.0;
	for(i=0; i<AXISCNT; i++)
	{
		if(B[5030+i*2]==1&&jogFlagVal[0+i*2]==0)
			edgeFlagVal[0+i*2]=1;
		if(B[5031+i*2]==1&&jogFlagVal[1+i*2]==0)
			edgeFlagVal[1+i*2]=1;
		if((UserDefSpeed>=GAPVALUE&&B[5030+i*2]==1&&SM[12]==0&&edgeFlagVal[0+i*2]==1)||
		        (UserDefSpeed<GAPVALUE&&B[5030+i*2]==0&&jogFlagVal[0+i*2]==1&&SM[RBRUN_ON_SM]==0))
		{
			if(SysModelType==1)//连续||单步
			{
				W[ERR_CODE_W]=27;
				return;
			}
			if(REF_COORD_INDEX==JOINT_COORD_INDEX)
				SM[JOINT_JOG_SM(i*2)]=1;
			else
				SM[COORD_JOG_SM(i*2)]=1;
		}
		else if((UserDefSpeed>=GAPVALUE&&B[5031+i*2]==1&&SM[12]==0&&edgeFlagVal[1+i*2]==1)||
		        (UserDefSpeed<GAPVALUE&&B[5031+i*2]==0&&jogFlagVal[1+i*2]==1&&SM[RBRUN_ON_SM]==0))
		{
			if(SysModelType==1)//连续||单步
			{
				W[ERR_CODE_W]=27;
				return;
			}
			if(REF_COORD_INDEX==JOINT_COORD_INDEX)
				SM[JOINT_JOG_SM((1+i*2))]=1;
			else
				SM[COORD_JOG_SM((1+i*2))]=1;
		}
		jogFlagVal[0+i*2]=B[5030+i*2];
		jogFlagVal[1+i*2]=B[5031+i*2];
		if(SM[JOINT_JOG_SM(i*2)]==1||SM[JOINT_JOG_SM(1+i*2)]==1||SM[COORD_JOG_SM((i*2))]==1||SM[COORD_JOG_SM((1+i*2))]==1)
		{
			if(REF_COORD_INDEX==JOINT_COORD_INDEX)//关节坐标系
			{
				AxisJogSpeed= (UserDefSpeed/100.0)*AxisJogSpeed_SET;
				if(AxisJogSpeed==0)
					AxisJogSpeed = 1;
				if(UserDefSpeed>=10)
					AxisJogStep = 1;
				else
					AxisJogStep = UserDefSpeed;
			}
			else
			{
				CoordJogSpeed= (UserDefSpeed/100.0)*CoordJogSpeed_SET;
				if(CoordJogSpeed==0)
					CoordJogSpeed=1;
				if(UserDefSpeed>=10)
					CoordJogStep = 1;
				else
					CoordJogStep = UserDefSpeed;
			}
			break;
		}
	}
}

void checkArea(WORD W,BIT B)
{
#define SysRegAddr_HD_SD_FD_SM_HSD_Y_X_HM
#define BASEPOINT_ADDR_HD 24000
#define AreaStatus_M 5100
#define AreaCheckEnable_HM 5000

	float basePos[6]= {0},curPos[6]={0};
	float lenth_X =  FHD[24012];
	float width_Y =  FHD[24014];
	float height_Z = FHD[24016];

	memcpy(basePos,HD+24000,12*2);
	memcpy(curPos,SD+4000,12*2);
	if(SM[ROBOT_ON_SM]==1&&HM[AreaCheckEnable_HM]==1)
	{
		float delt_X = curPos[0]-basePos[0];
		float delt_Y = curPos[1]-basePos[1];
		float delt_Z = curPos[2]-basePos[2];
		
		float x_Max,x_Min,y_Max,y_Min,z_Max,z_Min;
		if(lenth_X>0)
		{
			x_Min = basePos[0]; 
			x_Max = basePos[0]+lenth_X; 
		}
		else
		{
			x_Min = basePos[0]+lenth_X; 
			x_Max = basePos[0]; 
		}
		
		if(width_Y>0)
		{
			y_Min = basePos[1]; 
			y_Max = basePos[1]+width_Y; 
		}
		else
		{
			y_Min = basePos[1]+width_Y; 
			y_Max = basePos[1]; 
		}
		
		if(height_Z>0)
		{
			z_Min = basePos[2]; 
			z_Max = basePos[2]+height_Z; 
		}
		else
		{
			z_Min = basePos[2]+height_Z; 
			z_Max = basePos[2]; 
		}
		
		if((curPos[0]>=x_Min&&curPos[0]<=x_Max)&&(curPos[1]>=y_Min&&curPos[1]<=y_Max)&&(curPos[2]>=z_Min&&curPos[2]<=z_Max))
		{
			B[AreaStatus_M]=1;
			W[ERR_CODE_W]=29;		
		}
		else
		{
			B[AreaStatus_M]=0;		
		}
	}
	else if(HM[AreaCheckEnable_HM]==0)
	{
		B[AreaStatus_M]=0;		
	}
}


void round_area(WORD W,BIT B)// 球形
{
	#define SysRegAddr_HD_SD_FD_SM_HSD_Y_X_HM
	#define BASEPOINT_ADDR_HD 24000
	#define AreaCheckEnable_HM1 5001
	#define AreaStatus_M 5100
		float basePos[6]= {0},curPos[6]={0};
		float radius=FHD[24110];//半径设置。
		memcpy(basePos,HD+24000,12*2);//基准点
		memcpy(curPos,SD+4000,12*2);//当前点
		float x_sub;
		float y_sub;
		float z_sub;
		float sub_val;
		if(SM[ROBOT_ON_SM]==1&&HM[AreaCheckEnable_HM1]==1)
		{
			x_sub=curPos[0]-basePos[0];
			y_sub=curPos[1]-basePos[1];
			z_sub=curPos[2]-basePos[2];
			sub_val=x_sub*x_sub+y_sub*y_sub+z_sub*z_sub;
			radius=radius*radius;
			if(sub_val<=radius)
			{	
				B[AreaStatus_M]=1;
				W[ERR_CODE_W]=29;
			}
			else
				B[AreaStatus_M]=0;
		}
		else
			B[AreaStatus_M]=0;
}



void cylinder_area(WORD W,BIT B)//圆柱体
{	#define SysRegAddr_HD_SD_FD_SM_HSD_Y_X_HM
	#define AreaCheckEnable_HM2 5002
	#define AreaStatus_M 5100
		float basePos[6]= {0},curPos[6]={0};
		float radius=FHD[24112];//半径设置。
		float z_height=FHD[24114];//高度设置
		memcpy(basePos,HD+24000,12*2);//基准点
		memcpy(curPos,SD+4000,12*2);//当前点
		float x_sub;
		float y_sub;
		float z_sub;
		float sub_val;
		float z_Max,z_Min;
		if(SM[ROBOT_ON_SM]==1&&HM[AreaCheckEnable_HM2]==1)
		{
			x_sub=curPos[0]-basePos[0];
			y_sub=curPos[1]-basePos[1];
			sub_val=x_sub*x_sub+y_sub*y_sub;
			radius=radius*radius;
			if(z_height>0)
				{
					z_Max=z_height+basePos[2];
					z_Min=basePos[2];
				}
			else if(z_height<0)
			{
				z_Min=z_height+basePos[2];
				z_Max=basePos[2];
			}
			if(sub_val<=radius&&(curPos[2]>=z_Min&&curPos[2]<=z_Max))
			{
				B[AreaStatus_M]=1;
				W[ERR_CODE_W]=29;
			}
			else
				B[AreaStatus_M]=0;
		}
		else
			B[AreaStatus_M]=0;
}

C FUNCTION BLOCK tcrc.fcb
/* CRC校验生成
数据个数(n)输入:     W[0]
数据(整数)起始地址:  W[1]
...                  ...
数据(整数)结束地址:  W[n+1]
CRC校验结果存放地址：W[n+2]
W[n+3]
例:
TCRC D0 M0
数据个数: D0=0x06
数据输入: D1=0x01, D2=0x05, D3=0x48
D4=0x00, D5=0xFF, D6=0x00
结果显示: D7=0x9B, D8=0x9A */
/*************************************************************************
   FunctionBlockName:  TCRC
   Version:            1.0.0
   Author:             无锡信捷电气股份有限公司
   UpdateTime:         2010-4-22 10:01:36
   Comment:            
			CRC校验生成  
			
			数据个数(n)输入:     W[0] 
      数据(整数)起始地址:  W[1]
      ...                  ...
      数据(整数)结束地址:  W[n+1]
      CRC校验结果存放地址：W[n+2]
                           W[n+3]  
			例:
			TCRC D0 M0
			
			数据个数: D0=0x06
      数据输入: D1=0x01, D2=0x05, D3=0x48
                D4=0x00, D5=0xFF, D6=0x00
      结果显示: D7=0x9B, D8=0x9A
**************************************************************************/
void TCRC( WORD W , BIT B )
{
	int i,j,m,n;
	unsigned int crc_reg=0xffff,k;
	for (i=0;i<W[0];i++)
	{
		crc_reg^=W[i+1];
		for(j=0;j<8;j++)
		{
			if(crc_reg&0x01)
			   crc_reg=(crc_reg>>1)^0xa001;
			else
			   crc_reg=crc_reg>>1;
		}
	}
	
	m=W[0]+1;
	n=W[0]+2;
	k=crc_reg&0xff00;
	W[n]=k>>8;
	W[m]=crc_reg&0x00ff;
}